{attribute 'linkalways'} 
{attribute 'no_explicit_call' := 'This FB is a CLASS and must be accessed using methods or properties'}
{attribute 'enable_dynamic_creation'}
FUNCTION_BLOCK Node_F_VN_ConvertPolarToCartesianPointsExp EXTENDS VisionNode
VAR
	ipSrcPointsPolar : _ITcVnContainer;
    ipDestPointsCart : _ITcVnContainer;
    bAngleInDegrees : _BOOL(FALSE);
    hrPrev : _HRESULT(S_OK);
	hresult : _HRESULT(S_OK);
END_VAR

METHOD PUBLIC  Clone : I_Node
VAR
	pNode : POINTER TO Node_F_VN_ConvertPolarToCartesianPointsExp;
END_VAR
pNode := __NEW(Node_F_VN_ConvertPolarToCartesianPointsExp);
Clone := pNode^;
END_METHOD

METHOD FB_init : BOOL
VAR_INPUT
	bInitRetains : BOOL; // if TRUE, the retain variables are initialized (warm start / cold start)
	bInCopyCode : BOOL;  // if TRUE, the instance afterwards gets moved into the copy code (online change)
END_VAR
AddInput('ipSrcPointsPolar', ipSrcPointsPolar);
AddParameter('bAngleInDegrees', bAngleInDegrees);
AddInput('hrPrev', hrPrev);
AddOutput('ipDestPointsCart', ipDestPointsCart);
AddOutput('hresult',hresult);
END_METHOD

METHOD PROTECTED OnExecute
hresult.Value := F_VN_ConvertPolarToCartesianPointsExp(
	ipSrcPointsPolar := ipSrcPointsPolar.Value,
	ipDestPointsCart := ipDestPointsCart.Value,
    bAngleInDegrees := bAngleInDegrees.Value,
	hrPrev := hrPrev.Value);
END_METHOD

METHOD PUBLIC PreExecutionCheck
VAR_INPUT
	Check : I_PreExecutionChecks;
END_VAR
Check.IsTrue(ipSrcPointsPolar.IsValid, 'ipSrcPointsPolar must be a valid container');
Check.IsTrue((ipSrcPointsPolar.IsType(TC_GLOBAL_CONST_LIST.ContainerType_Vector_TcVnPoint2_REAL) OR
              ipSrcPointsPolar.IsType(TC_GLOBAL_CONST_LIST.ContainerType_Vector_TcVnPoint2_LREAL)),
              'ipSrcPointsPolar contains incorrect type');
END_METHOD

END_FUNCTION_BLOCK

(* stored: Version 1.1.0.1, ProductVersion 3.1.4026.13
   POU Node_F_VN_ConvertPolarToCartesianPointsExp: Id {63622d8e-239d-077a-3965-6eacd84452d8}, SpecialFunc None
   Folder Constructor: Id {d59a3f7e-1bf7-07c4-1e39-71a111d21519}
   Method Clone: Id {7d0b7cc7-a1f9-0ce2-10bb-c7a05b30a9da}
   Method FB_init: Id {19f8e871-51b1-09b9-2851-9cd4b36df041}
   Method OnExecute: Id {e5ae78a0-db5b-0bdb-28c4-eeb08b6e28b2}
   Method PreExecutionCheck: Id {0dbedac2-fefe-0331-2b2e-e38eebce7c1c} *)
